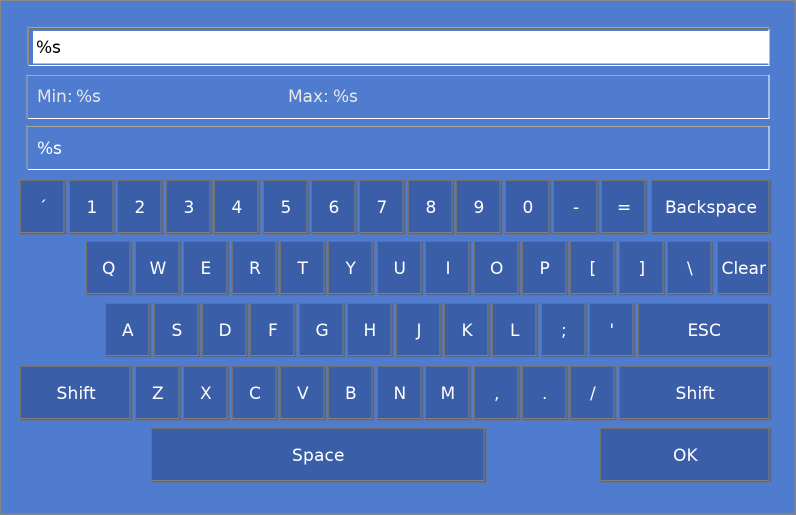
VISUALIZATION KlawiaturaLitery  // 796x515
VAR_INPUT
	stVariableValue : STRING;
	stMin : STRING;
	stMax : STRING;
	stTitle : STRING;
	flags : DWORD;
END_VAR
VAR
	bInit : BOOL;
	bShift : BOOL;
	stMessage : STRING;
	stOutputValue : STRING;
END_VAR
    Rectangle (0,0 796x515)
    Rectangle (12,169 773x70)
    Rectangle (12,240 773x62)
    Rectangle (12,301 773x63)
    Rectangle (12,364 773x62)
    Rectangle (12,423 773x75)
    Button (600,428 171x54), "OK"
        OnMouseDown: CloseDialog Dialog=KlawiaturaLitery, Result=OK, NumpadKeypad=True, NumpadKeypadSet=True
    Button (638,303 133x54), "ESC"
        OnMouseDown: CloseDialog Dialog=KlawiaturaLitery, Result=Cancel, NumpadKeypad=True, NumpadKeypadSet=True
    Button (717,241 54x54), "Clear"
        OnMouseDown: execute { stVariableValue := ''; stOutputValue := ''; }
    Button (651,180 120x54), "Backspace"
        OnMouseDown: execute { VisuDlg_CheckedBack(stOutputValue, stVariableValue, bInit); }
    Button (619,366 152x54), "Shift"
        OnMouseDown: toggle bShift
    Button (151,428 335x54), "Space"
        OnMouseDown: execute { VisuDlg_CheckedAppend(stOutputValue, stVariableValue, bInit, (flags AND VisuElems.Visu_InputFlags.Password) = 1, ' '); }
    Button (667,241 46x54), "|", invisible if: NOT bShift
        OnMouseDown: execute { VisuDlg_CheckedAppend(stOutputValue, stVariableValue, bInit, (flags AND VisuElems.Visu_InputFlags.Password) = 1, '|'); }
    Button (474,366 46x54), "<", invisible if: NOT bShift
        OnMouseDown: execute { VisuDlg_CheckedAppend(stOutputValue, stVariableValue, bInit, (flags AND VisuElems.Visu_InputFlags.Password) = 1, '<'); }
    Button (522,366 46x54), ">", invisible if: NOT bShift
        OnMouseDown: execute { VisuDlg_CheckedAppend(stOutputValue, stVariableValue, bInit, (flags AND VisuElems.Visu_InputFlags.Password) = 1, '>'); }
    Button (328,241 46x54), "y", invisible if: NOT bShift
        OnMouseDown: execute { VisuDlg_CheckedAppend(stOutputValue, stVariableValue, bInit, (flags AND VisuElems.Visu_InputFlags.Password) = 1, 'y'); }
    Button (328,241 46x54), "Y", invisible if: bShift
        OnMouseDown: execute { VisuDlg_CheckedAppend(stOutputValue, stVariableValue, bInit, (flags AND VisuElems.Visu_InputFlags.Password) = 1, 'Y'); }
    Button (183,366 46x54), "x", invisible if: NOT bShift
        OnMouseDown: execute { VisuDlg_CheckedAppend(stOutputValue, stVariableValue, bInit, (flags AND VisuElems.Visu_InputFlags.Password) = 1, 'x'); }
    Button (183,366 46x54), "X", invisible if: bShift
        OnMouseDown: execute { VisuDlg_CheckedAppend(stOutputValue, stVariableValue, bInit, (flags AND VisuElems.Visu_InputFlags.Password) = 1, 'X'); }
    Button (232,366 46x54), "c", invisible if: NOT bShift
        OnMouseDown: execute { VisuDlg_CheckedAppend(stOutputValue, stVariableValue, bInit, (flags AND VisuElems.Visu_InputFlags.Password) = 1, 'c'); }
    Button (232,366 46x54), "C", invisible if: bShift
        OnMouseDown: execute { VisuDlg_CheckedAppend(stOutputValue, stVariableValue, bInit, (flags AND VisuElems.Visu_InputFlags.Password) = 1, 'C'); }
    Button (280,366 46x54), "v", invisible if: NOT bShift
        OnMouseDown: execute { VisuDlg_CheckedAppend(stOutputValue, stVariableValue, bInit, (flags AND VisuElems.Visu_InputFlags.Password) = 1, 'v'); }
    Button (280,366 46x54), "V", invisible if: bShift
        OnMouseDown: execute { VisuDlg_CheckedAppend(stOutputValue, stVariableValue, bInit, (flags AND VisuElems.Visu_InputFlags.Password) = 1, 'V'); }
    Button (328,366 46x54), "b", invisible if: NOT bShift
        OnMouseDown: execute { VisuDlg_CheckedAppend(stOutputValue, stVariableValue, bInit, (flags AND VisuElems.Visu_InputFlags.Password) = 1, 'b'); }
    Button (328,366 46x54), "B", invisible if: bShift
        OnMouseDown: execute { VisuDlg_CheckedAppend(stOutputValue, stVariableValue, bInit, (flags AND VisuElems.Visu_InputFlags.Password) = 1, 'B'); }
    Button (377,366 46x54), "n", invisible if: NOT bShift
        OnMouseDown: execute { VisuDlg_CheckedAppend(stOutputValue, stVariableValue, bInit, (flags AND VisuElems.Visu_InputFlags.Password) = 1, 'n'); }
    Button (377,366 46x54), "N", invisible if: bShift
        OnMouseDown: execute { VisuDlg_CheckedAppend(stOutputValue, stVariableValue, bInit, (flags AND VisuElems.Visu_InputFlags.Password) = 1, 'N'); }
    Button (425,366 46x54), "m", invisible if: NOT bShift
        OnMouseDown: execute { VisuDlg_CheckedAppend(stOutputValue, stVariableValue, bInit, (flags AND VisuElems.Visu_InputFlags.Password) = 1, 'm'); }
    Button (425,366 46x54), "M", invisible if: bShift
        OnMouseDown: execute { VisuDlg_CheckedAppend(stOutputValue, stVariableValue, bInit, (flags AND VisuElems.Visu_InputFlags.Password) = 1, 'M'); }
    Button (541,303 46x54), ":", invisible if: NOT bShift
        OnMouseDown: execute { VisuDlg_CheckedAppend(stOutputValue, stVariableValue, bInit, (flags AND VisuElems.Visu_InputFlags.Password) = 1, ':'); }
    Button (553,180 46x54), "_", invisible if: NOT bShift
        OnMouseDown: execute { VisuDlg_CheckedAppend(stOutputValue, stVariableValue, bInit, (flags AND VisuElems.Visu_InputFlags.Password) = 1, '_'); }
    Button (105,303 46x54), "a", invisible if: NOT bShift
        OnMouseDown: execute { VisuDlg_CheckedAppend(stOutputValue, stVariableValue, bInit, (flags AND VisuElems.Visu_InputFlags.Password) = 1, 'a'); }
    Button (105,303 46x54), "A", invisible if: bShift
        OnMouseDown: execute { VisuDlg_CheckedAppend(stOutputValue, stVariableValue, bInit, (flags AND VisuElems.Visu_InputFlags.Password) = 1, 'A'); }
    Button (154,303 46x54), "s", invisible if: NOT bShift
        OnMouseDown: execute { VisuDlg_CheckedAppend(stOutputValue, stVariableValue, bInit, (flags AND VisuElems.Visu_InputFlags.Password) = 1, 's'); }
    Button (154,303 46x54), "S", invisible if: bShift
        OnMouseDown: execute { VisuDlg_CheckedAppend(stOutputValue, stVariableValue, bInit, (flags AND VisuElems.Visu_InputFlags.Password) = 1, 'S'); }
    Button (202,303 46x54), "d", invisible if: NOT bShift
        OnMouseDown: execute { VisuDlg_CheckedAppend(stOutputValue, stVariableValue, bInit, (flags AND VisuElems.Visu_InputFlags.Password) = 1, 'd'); }
    Button (202,303 46x54), "D", invisible if: bShift
        OnMouseDown: execute { VisuDlg_CheckedAppend(stOutputValue, stVariableValue, bInit, (flags AND VisuElems.Visu_InputFlags.Password) = 1, 'D'); }
    Button (250,303 46x54), "f", invisible if: NOT bShift
        OnMouseDown: execute { VisuDlg_CheckedAppend(stOutputValue, stVariableValue, bInit, (flags AND VisuElems.Visu_InputFlags.Password) = 1, 'f'); }
    Button (250,303 46x54), "F", invisible if: bShift
        OnMouseDown: execute { VisuDlg_CheckedAppend(stOutputValue, stVariableValue, bInit, (flags AND VisuElems.Visu_InputFlags.Password) = 1, 'F'); }
    Button (299,303 46x54), "g", invisible if: NOT bShift
        OnMouseDown: execute { VisuDlg_CheckedAppend(stOutputValue, stVariableValue, bInit, (flags AND VisuElems.Visu_InputFlags.Password) = 1, 'g'); }
    Button (299,303 46x54), "G", invisible if: bShift
        OnMouseDown: execute { VisuDlg_CheckedAppend(stOutputValue, stVariableValue, bInit, (flags AND VisuElems.Visu_InputFlags.Password) = 1, 'G'); }
    Button (347,303 46x54), "h", invisible if: NOT bShift
        OnMouseDown: execute { VisuDlg_CheckedAppend(stOutputValue, stVariableValue, bInit, (flags AND VisuElems.Visu_InputFlags.Password) = 1, 'h'); }
    Button (347,303 46x54), "H", invisible if: bShift
        OnMouseDown: execute { VisuDlg_CheckedAppend(stOutputValue, stVariableValue, bInit, (flags AND VisuElems.Visu_InputFlags.Password) = 1, 'H'); }
    Button (396,303 46x54), "j", invisible if: NOT bShift
        OnMouseDown: execute { VisuDlg_CheckedAppend(stOutputValue, stVariableValue, bInit, (flags AND VisuElems.Visu_InputFlags.Password) = 1, 'j'); }
    Button (396,303 46x54), "J", invisible if: bShift
        OnMouseDown: execute { VisuDlg_CheckedAppend(stOutputValue, stVariableValue, bInit, (flags AND VisuElems.Visu_InputFlags.Password) = 1, 'J'); }
    Button (444,303 46x54), "k", invisible if: NOT bShift
        OnMouseDown: execute { VisuDlg_CheckedAppend(stOutputValue, stVariableValue, bInit, (flags AND VisuElems.Visu_InputFlags.Password) = 1, 'k'); }
    Button (444,303 46x54), "K", invisible if: bShift
        OnMouseDown: execute { VisuDlg_CheckedAppend(stOutputValue, stVariableValue, bInit, (flags AND VisuElems.Visu_InputFlags.Password) = 1, 'K'); }
    Button (492,303 46x54), "l", invisible if: NOT bShift
        OnMouseDown: execute { VisuDlg_CheckedAppend(stOutputValue, stVariableValue, bInit, (flags AND VisuElems.Visu_InputFlags.Password) = 1, 'l'); }
    Button (492,303 46x54), "L", invisible if: bShift
        OnMouseDown: execute { VisuDlg_CheckedAppend(stOutputValue, stVariableValue, bInit, (flags AND VisuElems.Visu_InputFlags.Password) = 1, 'L'); }
    Button (166,180 46x54), "#", invisible if: NOT bShift
        OnMouseDown: execute { VisuDlg_CheckedAppend(stOutputValue, stVariableValue, bInit, (flags AND VisuElems.Visu_InputFlags.Password) = 1, '#'); }
    Button (117,180 46x54), "@", invisible if: NOT bShift
        OnMouseDown: execute { VisuDlg_CheckedAppend(stOutputValue, stVariableValue, bInit, (flags AND VisuElems.Visu_InputFlags.Password) = 1, '@'); }
    Button (86,241 46x54), "q", invisible if: NOT bShift
        OnMouseDown: execute { VisuDlg_CheckedAppend(stOutputValue, stVariableValue, bInit, (flags AND VisuElems.Visu_InputFlags.Password) = 1, 'q'); }
    Button (86,241 46x54), "Q", invisible if: bShift
        OnMouseDown: execute { VisuDlg_CheckedAppend(stOutputValue, stVariableValue, bInit, (flags AND VisuElems.Visu_InputFlags.Password) = 1, 'Q'); }
    Button (135,241 46x54), "w", invisible if: NOT bShift
        OnMouseDown: execute { VisuDlg_CheckedAppend(stOutputValue, stVariableValue, bInit, (flags AND VisuElems.Visu_InputFlags.Password) = 1, 'w'); }
    Button (135,241 46x54), "W", invisible if: bShift
        OnMouseDown: execute { VisuDlg_CheckedAppend(stOutputValue, stVariableValue, bInit, (flags AND VisuElems.Visu_InputFlags.Password) = 1, 'W'); }
    Button (183,241 46x54), "e", invisible if: NOT bShift
        OnMouseDown: execute { VisuDlg_CheckedAppend(stOutputValue, stVariableValue, bInit, (flags AND VisuElems.Visu_InputFlags.Password) = 1, 'e'); }
    Button (183,241 46x54), "E", invisible if: bShift
        OnMouseDown: execute { VisuDlg_CheckedAppend(stOutputValue, stVariableValue, bInit, (flags AND VisuElems.Visu_InputFlags.Password) = 1, 'E'); }
    Button (232,241 46x54), "r", invisible if: NOT bShift
        OnMouseDown: execute { VisuDlg_CheckedAppend(stOutputValue, stVariableValue, bInit, (flags AND VisuElems.Visu_InputFlags.Password) = 1, 'r'); }
    Button (232,241 46x54), "R", invisible if: bShift
        OnMouseDown: execute { VisuDlg_CheckedAppend(stOutputValue, stVariableValue, bInit, (flags AND VisuElems.Visu_InputFlags.Password) = 1, 'R'); }
    Button (280,241 46x54), "t", invisible if: NOT bShift
        OnMouseDown: execute { VisuDlg_CheckedAppend(stOutputValue, stVariableValue, bInit, (flags AND VisuElems.Visu_InputFlags.Password) = 1, 't'); }
    Button (280,241 46x54), "T", invisible if: bShift
        OnMouseDown: execute { VisuDlg_CheckedAppend(stOutputValue, stVariableValue, bInit, (flags AND VisuElems.Visu_InputFlags.Password) = 1, 'T'); }
    Button (135,366 46x54), "z", invisible if: NOT bShift
        OnMouseDown: execute { VisuDlg_CheckedAppend(stOutputValue, stVariableValue, bInit, (flags AND VisuElems.Visu_InputFlags.Password) = 1, 'z'); }
    Button (135,366 46x54), "Z", invisible if: bShift
        OnMouseDown: execute { VisuDlg_CheckedAppend(stOutputValue, stVariableValue, bInit, (flags AND VisuElems.Visu_InputFlags.Password) = 1, 'Z'); }
    Button (377,241 46x54), "u", invisible if: NOT bShift
        OnMouseDown: execute { VisuDlg_CheckedAppend(stOutputValue, stVariableValue, bInit, (flags AND VisuElems.Visu_InputFlags.Password) = 1, 'u'); }
    Button (377,241 46x54), "U", invisible if: bShift
        OnMouseDown: execute { VisuDlg_CheckedAppend(stOutputValue, stVariableValue, bInit, (flags AND VisuElems.Visu_InputFlags.Password) = 1, 'U'); }
    Button (425,241 46x54), "i", invisible if: NOT bShift
        OnMouseDown: execute { VisuDlg_CheckedAppend(stOutputValue, stVariableValue, bInit, (flags AND VisuElems.Visu_InputFlags.Password) = 1, 'i'); }
    Button (425,241 46x54), "I", invisible if: bShift
        OnMouseDown: execute { VisuDlg_CheckedAppend(stOutputValue, stVariableValue, bInit, (flags AND VisuElems.Visu_InputFlags.Password) = 1, 'I'); }
    Button (474,241 46x54), "o", invisible if: NOT bShift
        OnMouseDown: execute { VisuDlg_CheckedAppend(stOutputValue, stVariableValue, bInit, (flags AND VisuElems.Visu_InputFlags.Password) = 1, 'o'); }
    Button (474,241 46x54), "O", invisible if: bShift
        OnMouseDown: execute { VisuDlg_CheckedAppend(stOutputValue, stVariableValue, bInit, (flags AND VisuElems.Visu_InputFlags.Password) = 1, 'O'); }
    Button (522,241 46x54), "p", invisible if: NOT bShift
        OnMouseDown: execute { VisuDlg_CheckedAppend(stOutputValue, stVariableValue, bInit, (flags AND VisuElems.Visu_InputFlags.Password) = 1, 'p'); }
    Button (522,241 46x54), "P", invisible if: bShift
        OnMouseDown: execute { VisuDlg_CheckedAppend(stOutputValue, stVariableValue, bInit, (flags AND VisuElems.Visu_InputFlags.Password) = 1, 'P'); }
    Button (601,180 46x54), "+", invisible if: NOT bShift
        OnMouseDown: execute { VisuDlg_CheckedAppend(stOutputValue, stVariableValue, bInit, (flags AND VisuElems.Visu_InputFlags.Password) = 1, '+'); }
    Button (408,180 46x54), "*", invisible if: NOT bShift
        OnMouseDown: execute { VisuDlg_CheckedAppend(stOutputValue, stVariableValue, bInit, (flags AND VisuElems.Visu_InputFlags.Password) = 1, '*'); }
    Button (20,180 46x54), "~", invisible if: NOT bShift
        OnMouseDown: execute { VisuDlg_CheckedAppend(stOutputValue, stVariableValue, bInit, (flags AND VisuElems.Visu_InputFlags.Password) = 1, '~'); }
    Button (311,180 46x54), "^", invisible if: NOT bShift
        OnMouseDown: execute { VisuDlg_CheckedAppend(stOutputValue, stVariableValue, bInit, (flags AND VisuElems.Visu_InputFlags.Password) = 1, '^'); }
    Button (69,180 46x54), "!", invisible if: NOT bShift
        OnMouseDown: execute { VisuDlg_CheckedAppend(stOutputValue, stVariableValue, bInit, (flags AND VisuElems.Visu_InputFlags.Password) = 1, '!'); }
    Button (589,303 46x54), """, invisible if: NOT bShift
        OnMouseDown: execute { VisuDlg_CheckedAppend(stOutputValue, stVariableValue, bInit, (flags AND VisuElems.Visu_InputFlags.Password) = 1, '"'); }
    Button (214,180 46x54), "$", invisible if: NOT bShift
        OnMouseDown: execute { VisuDlg_CheckedAppend(stOutputValue, stVariableValue, bInit, (flags AND VisuElems.Visu_InputFlags.Password) = 1, '$$'); }
    Button (263,180 46x54), "%", invisible if: NOT bShift
        OnMouseDown: execute { VisuDlg_CheckedAppend(stOutputValue, stVariableValue, bInit, (flags AND VisuElems.Visu_InputFlags.Password) = 1, '%'); }
    Button (359,180 46x54), "&", invisible if: NOT bShift
        OnMouseDown: execute { VisuDlg_CheckedAppend(stOutputValue, stVariableValue, bInit, (flags AND VisuElems.Visu_InputFlags.Password) = 1, '&'); }
    Button (456,180 46x54), "(", invisible if: NOT bShift
        OnMouseDown: execute { VisuDlg_CheckedAppend(stOutputValue, stVariableValue, bInit, (flags AND VisuElems.Visu_InputFlags.Password) = 1, '('); }
    Button (505,180 46x54), ")", invisible if: NOT bShift
        OnMouseDown: execute { VisuDlg_CheckedAppend(stOutputValue, stVariableValue, bInit, (flags AND VisuElems.Visu_InputFlags.Password) = 1, ')'); }
    Button (570,366 46x54), "?", invisible if: NOT bShift
        OnMouseDown: execute { VisuDlg_CheckedAppend(stOutputValue, stVariableValue, bInit, (flags AND VisuElems.Visu_InputFlags.Password) = 1, '?'); }
    Rectangle (12,72 773x97)
    Rectangle (34,132 734x32), "%s", text variable: stMessage
    Rectangle (12,10 773x62)
    Polyline (27,169) (27,126) (769,126)
    Polyline (27,118) (27,75) (769,75)
    Polyline (28,65) (28,27) (769,27)
    Polyline (28,169) (769,169) (769,126)
    Polyline (28,118) (769,118) (769,75)
    Polyline (29,65) (769,65) (769,28)
    Polyline (29,63) (29,28) (769,28)
    Rectangle (33,31 736x32), "%s", text variable: stOutputValue
    Rectangle (34,80 42x32), "Min:", text variable: stMin, invisible if: LEN(stMin) = 0
    Rectangle (73,80 157x32), "%s", text variable: stMin, invisible if: LEN(stMin) = 0
    Rectangle (285,80 45x32), "Max:", text variable: stMin, invisible if: LEN(stMax) = 0
    Rectangle (330,80 217x32), "%s", text variable: stMax, invisible if: LEN(stMax) = 0
    Button (20,180 46x54), "´", invisible if: bShift
        OnMouseDown: execute { VisuDlg_CheckedAppend(stOutputValue, stVariableValue, bInit, (flags AND VisuElems.Visu_InputFlags.Password) = 1, '´'); }
    Button (69,180 46x54), "1", invisible if: bShift
        OnMouseDown: execute { VisuDlg_CheckedAppend(stOutputValue, stVariableValue, bInit, (flags AND VisuElems.Visu_InputFlags.Password) = 1, '1'); }
    Button (117,180 46x54), "2", invisible if: bShift
        OnMouseDown: execute { VisuDlg_CheckedAppend(stOutputValue, stVariableValue, bInit, (flags AND VisuElems.Visu_InputFlags.Password) = 1, '2'); }
    Button (166,180 46x54), "3", invisible if: bShift
        OnMouseDown: execute { VisuDlg_CheckedAppend(stOutputValue, stVariableValue, bInit, (flags AND VisuElems.Visu_InputFlags.Password) = 1, '3'); }
    Button (214,180 46x54), "4", invisible if: bShift
        OnMouseDown: execute { VisuDlg_CheckedAppend(stOutputValue, stVariableValue, bInit, (flags AND VisuElems.Visu_InputFlags.Password) = 1, '4'); }
    Button (263,180 46x54), "5", invisible if: bShift
        OnMouseDown: execute { VisuDlg_CheckedAppend(stOutputValue, stVariableValue, bInit, (flags AND VisuElems.Visu_InputFlags.Password) = 1, '5'); }
    Button (311,180 46x54), "6", invisible if: bShift
        OnMouseDown: execute { VisuDlg_CheckedAppend(stOutputValue, stVariableValue, bInit, (flags AND VisuElems.Visu_InputFlags.Password) = 1, '6'); }
    Button (359,180 46x54), "7", invisible if: bShift
        OnMouseDown: execute { VisuDlg_CheckedAppend(stOutputValue, stVariableValue, bInit, (flags AND VisuElems.Visu_InputFlags.Password) = 1, '7'); }
    Button (408,180 46x54), "8", invisible if: bShift
        OnMouseDown: execute { VisuDlg_CheckedAppend(stOutputValue, stVariableValue, bInit, (flags AND VisuElems.Visu_InputFlags.Password) = 1, '8'); }
    Button (456,180 46x54), "9", invisible if: bShift
        OnMouseDown: execute { VisuDlg_CheckedAppend(stOutputValue, stVariableValue, bInit, (flags AND VisuElems.Visu_InputFlags.Password) = 1, '9'); }
    Button (505,180 46x54), "0", invisible if: bShift
        OnMouseDown: execute { VisuDlg_CheckedAppend(stOutputValue, stVariableValue, bInit, (flags AND VisuElems.Visu_InputFlags.Password) = 1, '0'); }
    Button (553,180 46x54), "-", invisible if: bShift
        OnMouseDown: execute { VisuDlg_CheckedAppend(stOutputValue, stVariableValue, bInit, (flags AND VisuElems.Visu_InputFlags.Password) = 1, '-'); }
    Button (601,180 46x54), "=", invisible if: bShift
        OnMouseDown: execute { VisuDlg_CheckedAppend(stOutputValue, stVariableValue, bInit, (flags AND VisuElems.Visu_InputFlags.Password) = 1, '='); }
    Button (570,241 46x54), "{", invisible if: NOT bShift
        OnMouseDown: execute { VisuDlg_CheckedAppend(stOutputValue, stVariableValue, bInit, (flags AND VisuElems.Visu_InputFlags.Password) = 1, '{'); }
    Button (570,241 46x54), "[", invisible if: bShift
        OnMouseDown: execute { VisuDlg_CheckedAppend(stOutputValue, stVariableValue, bInit, (flags AND VisuElems.Visu_InputFlags.Password) = 1, '['); }
    Button (619,241 46x54), "}", invisible if: NOT bShift
        OnMouseDown: execute { VisuDlg_CheckedAppend(stOutputValue, stVariableValue, bInit, (flags AND VisuElems.Visu_InputFlags.Password) = 1, '}'); }
    Button (619,241 46x54), "]", invisible if: bShift
        OnMouseDown: execute { VisuDlg_CheckedAppend(stOutputValue, stVariableValue, bInit, (flags AND VisuElems.Visu_InputFlags.Password) = 1, ']'); }
    Button (667,241 46x54), "\", invisible if: bShift
        OnMouseDown: execute { VisuDlg_CheckedAppend(stOutputValue, stVariableValue, bInit, (flags AND VisuElems.Visu_InputFlags.Password) = 1, '\'); }
    Button (541,303 46x54), ";", invisible if: bShift
        OnMouseDown: execute { VisuDlg_CheckedAppend(stOutputValue, stVariableValue, bInit, (flags AND VisuElems.Visu_InputFlags.Password) = 1, ';'); }
    Button (589,303 46x54), "'", invisible if: bShift
        OnMouseDown: execute { VisuDlg_CheckedAppend(stOutputValue, stVariableValue, bInit, (flags AND VisuElems.Visu_InputFlags.Password) = 1, '$''); }
    Button (474,366 46x54), ",", invisible if: bShift
        OnMouseDown: execute { VisuDlg_CheckedAppend(stOutputValue, stVariableValue, bInit, (flags AND VisuElems.Visu_InputFlags.Password) = 1, ','); }
    Button (522,366 46x54), ".", invisible if: bShift
        OnMouseDown: execute { VisuDlg_CheckedAppend(stOutputValue, stVariableValue, bInit, (flags AND VisuElems.Visu_InputFlags.Password) = 1, '.'); }
    Button (570,366 46x54), "/", invisible if: bShift
        OnMouseDown: execute { VisuDlg_CheckedAppend(stOutputValue, stVariableValue, bInit, (flags AND VisuElems.Visu_InputFlags.Password) = 1, '/'); }
    Button (20,366 112x54), "Shift"
        OnMouseDown: toggle bShift
END_VISUALIZATION

(* stored: Version 1.1.0.1
   Visu KlawiaturaLitery: Id {c2cc9e9c-7c80-482f-a39f-157c2a752e22} *)
